ABB RobotStudio station: HuiswerkOpdrachten.rsstnx

Station HuiswerkOpdrachten (saved by RobotStudio 23.3.10550.0)
Controller IRB120_3_58_1
  mechanical unit ROB_1: IRB120_3_58__01, 6 joints, base frame (0, 0, 0) mm
Layout (positions relative to the parent item):
  - tTrainingTool [mechanism] at (86.93, 218.99, 406.62) mm, rotated rx -178.74 ry 68.21 rz -178.69 deg
      TCP tTrainingTool at (31.79, 0, 229.64) mm, rotated rx 0 ry 38 rz 0 deg
      links: SpintecTool
  - IRB120_3_58__01 [mechanism, from %ABB.RobotStudio.Models.IRB120%\IRB120_3_58_G_01.rslib] at (0, 0, 0) mm; joint values [1.4794, -0.2491, 0.8685, -1.3033, 1.2831, 2.125] (rad or m)
  - Curve_thing_2 [part, from Training Objects\Curve_Thing.rslib] at (194.62, 412.46, 199.75) mm, rotated rx -0.1 ry -0.04 rz -89.23 deg
  - Table [part] at (200, 112.5, 0) mm, size 250 x 375 x 200 mm
  - Frame_1 [frame] at (31.79, 0, 229.64) mm, rotated rx 0 ry 38 rz 0 deg
Attachment: tTrainingTool is attached to IRB120_3_58__01 / Link6
Attachment: wTable is attached to Table
Attachment: wCurveThing is attached to Curve_thing_2
Attachment: Curve_thing_2 is attached to Table
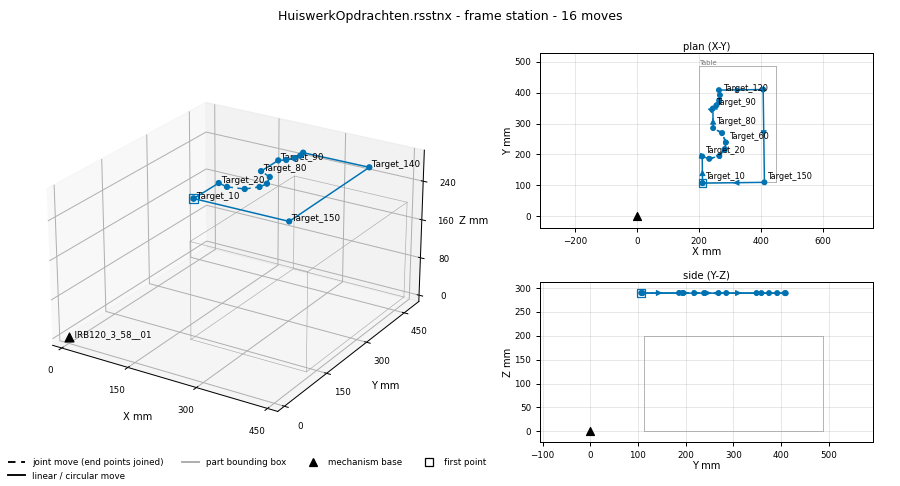
[picture p0: tool path of HuiswerkOpdrachten.rsstnx in frame station, 16 of 17 moves have a stored position in this frame; points joined in program order, loops and branches not executed]
Targets, tools, work objects and paths stored in the station, written as RAPID:
! task T_ROB1
MODULE CalibData
  PERS tooldata tTrainingTool:=[TRUE,[[31.793,0,229.639],[0.945518576,0,0.325568154,0]],[3,[-54.486,0,119.208],[1,0,0,0],0,0,0]];
  TASK PERS wobjdata wTable:=[FALSE,TRUE,"",[[200,112.5,200],[1,0,0,0]],[[0,0,0],[1,0,0,0]]];
  TASK PERS wobjdata wCurveThing:=[FALSE,TRUE,"",[[200.153881695,12.559984954,290.000001931],[0.99997695,-0.000323307,0.000861179,0.006727109]],[[0,0,0],[1,0,0,0]]];
ENDMODULE

! task T_ROB1
MODULE MainModule
  CONST robtarget Target_10:=[[13.339457543,94.549134052,0.00304146],[0.2000503,-0.728111971,-0.629237448,-0.184100703],[0,-1,1,0],[9E+09,9E+09,9E+09,9E+09,9E+09,9E+09]];
  CONST robtarget Target_20:=[[13.332826218,181.017070199,-0.002085504],[0.208470218,-0.0367133,0.938401725,-0.273119946],[1,-1,1,0],[9E+09,9E+09,9E+09,9E+09,9E+09,9E+09]];
  CONST robtarget Target_40:=[[68.886844506,181.679741052,0.004277473],[0.20763609,-0.040383239,0.933538766,-0.289416344],[0,-1,1,0],[9E+09,9E+09,9E+09,9E+09,9E+09,9E+09]];
  CONST robtarget Target_50:=[[86.992032728,204.238232069,-0.000542538],[0.248142733,0.022796746,0.968448604,-0.003576738],[0,-1,1,0],[9E+09,9E+09,9E+09,9E+09,9E+09,9E+09]];
  CONST robtarget Target_30:=[[36.028653379,173.130972729,0.101493998],[0.192176514,0.008539127,0.934406114,-0.299800743],[1,-1,1,0],[9E+09,9E+09,9E+09,9E+09,9E+09,9E+09]];
  CONST robtarget Target_60:=[[90.570786944,224.931972594,-0.001231747],[0.314788255,-0.103404198,0.936171663,0.117467202],[0,-2,1,0],[9E+09,9E+09,9E+09,9E+09,9E+09,9E+09]];
  CONST robtarget Target_70:=[[78.511692534,255.547076122,-0.002261983],[0.29266045,-0.161496995,0.929053949,0.158516062],[0,-2,1,0],[9E+09,9E+09,9E+09,9E+09,9E+09,9E+09]];
  CONST robtarget Target_80:=[[50.000767435,272.032034665,-0.000958088],[0.256842653,-0.038605415,0.951258076,0.16628153],[1,-1,1,0],[9E+09,9E+09,9E+09,9E+09,9E+09,9E+09]];
  CONST robtarget Target_90:=[[50.004134212,335.457537805,-0.000775987],[0.303506126,0.382546019,0.871854043,0.037591258],[0,-1,1,0],[9E+09,9E+09,9E+09,9E+09,9E+09,9E+09]];
  CONST robtarget Target_100:=[[61.600998929,345.552637331,-0.004439553],[0.319393216,0.369031587,0.872813351,-0.000717926],[0,-1,1,0],[9E+09,9E+09,9E+09,9E+09,9E+09,9E+09]];
  CONST robtarget Target_110:=[[70.615208711,361.412818585,0.001383803],[0.319393434,0.369057732,0.87280218,-0.000761067],[0,-1,1,0],[9E+09,9E+09,9E+09,9E+09,9E+09,9E+09]];
  CONST robtarget Target_120:=[[73.35479978,378.457518754,-0.003354051],[0.3026277,0.064615344,0.945337596,0.10285019],[1,-1,1,0],[9E+09,9E+09,9E+09,9E+09,9E+09,9E+09]];
  CONST robtarget Target_130:=[[70.461044386,394.547866855,0.001970142],[0.319174324,0.330611414,0.888060707,0.01311581],[0,-1,1,0],[9E+09,9E+09,9E+09,9E+09,9E+09,9E+09]];
  CONST robtarget Target_140:=[[213.334289144,394.555724872,-0.001120603],[0.008745743,0.340533424,-0.920943807,0.189269658],[0,-1,0,0],[9E+09,9E+09,9E+09,9E+09,9E+09,9E+09]];
  CONST robtarget Target_150:=[[213.337859733,94.548493566,-0.001634481],[0.263393572,-0.331833974,-0.903578019,-0.063693041],[0,-1,0,0],[9E+09,9E+09,9E+09,9E+09,9E+09,9E+09]];
  CONST robtarget Target_160:=[[13.339442446,94.549137974,0.003048941],[0.174490808,0.006681271,0.984635768,-0.000849953],[1,-1,1,0],[9E+09,9E+09,9E+09,9E+09,9E+09,9E+09]];
  CONST jointtarget JointTarget_1:=[[0,0,0,0,0,0],[9E+09,9E+09,9E+09,9E+09,9E+09,9E+09]];
  PROC Path_20()
    MoveJ Target_10,v50,z100,tTrainingTool\WObj:=wCurveThing;
    MoveL Target_20,v50,fine,tTrainingTool\WObj:=wCurveThing;
    MoveJ Target_30,v50,z100,tTrainingTool\WObj:=wCurveThing;
    MoveJ Target_40,v50,z100,tTrainingTool\WObj:=wCurveThing;
    MoveJ Target_50,v50,z100,tTrainingTool\WObj:=wCurveThing;
    MoveJ Target_60,v50,z100,tTrainingTool\WObj:=wCurveThing;
    MoveJ Target_70,v50,z100,tTrainingTool\WObj:=wCurveThing;
    MoveJ Target_80,v50,z100,tTrainingTool\WObj:=wCurveThing;
    MoveL Target_90,v50,fine,tTrainingTool\WObj:=wCurveThing;
    MoveJ Target_100,v50,z100,tTrainingTool\WObj:=wCurveThing;
    MoveJ Target_110,v50,z100,tTrainingTool\WObj:=wCurveThing;
    MoveJ Target_120,v50,z100,tTrainingTool\WObj:=wCurveThing;
    MoveJ Target_130,v50,z100,tTrainingTool\WObj:=wCurveThing;
    MoveL Target_140,v50,fine,tTrainingTool\WObj:=wCurveThing;
    MoveL Target_150,v50,fine,tTrainingTool\WObj:=wCurveThing;
    MoveL Target_160,v50,z100,tTrainingTool\WObj:=wCurveThing;
  ENDPROC
  PROC Path_30()
    MoveAbsJ JointTarget_1,v1000,z100,tTrainingTool\WObj:=wCurveThing;
  ENDPROC
ENDMODULE

